// TIA Portal V17 export
// export: Created 2023-02-13T11:05:56.0459047Z, ExportSetting WithDefaults, DisplayName Totally Integrated Automation Portal, DisplayVersion V17, DisplayName TIA Portal Openness, DisplayVersion V17, DisplayName TIA Portal Teamcenter Gateway, DisplayVersion V17, DisplayName TIA Portal Version Control Interface, DisplayVersion V17, DisplayName SINAMICS Startdrive Advanced, DisplayVersion V17, DisplayName SINAMICS Startdrive G130, G150, S120, S150, SINAMICS MV, S210, DisplayVersion V17, DisplayName SINAMICS Startdrive G110M, G120, G120C, G120D, G120P, G115D, DisplayVersion V17, DisplayName STEP 7 Professional, DisplayVersion V17, DisplayName STEP 7 Safety, DisplayVersion V17, DisplayName WinCC Professional, DisplayVersion V17
VAR_GLOBAL   // PLC tag table "Tag table_1"
   "FT-02.01_Mass flow Value" AT %ID115 : Real;
   "FT-02.01_Mass flow Status" AT %IB119 : Byte;
   "FT-02.01_Volume flow Value" AT %ID120 : Real;
   "FT-02.01_Volume flow Status" AT %IB124 : Byte;
   "FT-02.01_Corrected volume flow Value" AT %ID125 : Real;
   "FT-02.01_Corrected volume flow Status" AT %IB129 : Byte;
   "FT-02.01_Density Value" AT %ID130 : Real;
   "FT-02.01_Density Status" AT %IB134 : Byte;
   "FT-02.01_Reference Density Value" AT %ID135 : Real;
   "FT-02.01_Reference Density Status" AT %IB139 : Byte;
   "FT-02.01_Temperature Value" AT %ID140 : Real;
   "FT-02.01_Temperature Status" AT %IB144 : Byte;
   "FT-02.01_Totalizer_1 Value" AT %ID145 : Real;
   "FT-02.01_Totalizer_1 Status" AT %IB149 : Byte;
   "FT-02.01_Totalizer_2 Value" AT %ID150 : Real;
   "FT-02.01_Totalizer_2 Status" AT %IB154 : Byte;
   "FT-02.01_Totalizer_3 Value" AT %ID155 : Real;
   "FT-02.01_Totalizer_3 Status" AT %IB159 : Byte;
   "FT-03.01_Mass flow Value" AT %ID160 : Real;
   "FT-03.01_Mass flow Status" AT %IB164 : Byte;
   "FT-03.01_Volume flow Value" AT %ID165 : Real;
   "FT-03.01_Volume flow Status" AT %IB169 : Byte;
   "FT-03.01_Corrected volume flow Value" AT %ID170 : Real;
   "FT-03.01_Corrected volume flow Status" AT %IB174 : Byte;
   "FT-03.01_Density Value" AT %ID175 : Real;
   "FT-03.01_Density Status" AT %IB179 : Byte;
   "FT-03.01_Reference Density Value" AT %ID180 : Real;
   "FT-03.01_Reference Density Status" AT %IB184 : Byte;
   "FT-03.01_Temperature Value" AT %ID185 : Real;
   "FT-03.01_Temperature Status" AT %IB189 : Byte;
   "FT-03.01_Totalizer_1 Value" AT %ID190 : Real;
   "FT-03.01_Totalizer_1 Status" AT %IB194 : Byte;
   "FT-03.01_Totalizer_2 Value" AT %ID195 : Real;
   "FT-03.01_Totalizer_2 Status" AT %IB199 : Byte;
   "FT-03.01_Totalizer_3 Value" AT %ID200 : Real;
   "FT-03.01_Totalizer_3 Status" AT %IB204 : Byte;
   "FT-04.01_Mass flow Value" AT %ID205 : Real;
   "FT-04.01_Mass flow Status" AT %IB209 : Byte;
   "FT-04.01_Volume flow Value" AT %ID210 : Real;
   "FT-04.01_Volume flow Status" AT %IB214 : Byte;
   "FT-04.01_Corrected volume flow Value" AT %ID215 : Real;
   "FT-04.01_Corrected volume flow Status" AT %IB219 : Byte;
   "FT-04.01_Density Value" AT %ID220 : Real;
   "FT-04.01_Density Status" AT %IB224 : Byte;
   "FT-04.01_Reference Density Value" AT %ID225 : Real;
   "FT-04.01_Reference Density Status" AT %IB229 : Byte;
   "FT-04.01_Temperature Value" AT %ID230 : Real;
   "FT-04.01_Temperature Status" AT %IB234 : Byte;
   "FT-04.01_Totalizer_1 Value" AT %ID235 : Real;
   "FT-04.01_Totalizer_1 Status" AT %IB239 : Byte;
   "FT-04.01_Totalizer_2 Value" AT %ID240 : Real;
   "FT-04.01_Totalizer_2 Status" AT %IB244 : Byte;
   "FT-04.01_Totalizer_3 Value" AT %ID245 : Real;
   "FT-04.01_Totalizer_3 Status" AT %IB249 : Byte;
   "FT-05.01_Mass flow Value" AT %ID250 : Real;
   "FT-05.01_Mass flow Status" AT %IB254 : Byte;
   "FT-05.01_Volume flow Value" AT %ID255 : Real;
   "FT-05.01_Volume flow Status" AT %IB259 : Byte;
   "FT-05.01_Corrected volume flow Value" AT %ID260 : Real;
   "FT-05.01_Corrected volume flow Status" AT %IB264 : Byte;
   "FT-05.01_Density Value" AT %ID265 : Real;
   "FT-05.01_Density Status" AT %IB269 : Byte;
   "FT-05.01_Reference Density Value" AT %ID270 : Real;
   "FT-05.01_Reference Density Status" AT %IB274 : Byte;
   "FT-05.01_Temperature Value" AT %ID275 : Real;
   "FT-05.01_Temperature Status" AT %IB279 : Byte;
   "FT-05.01_Totalizer_1 Value" AT %ID280 : Real;
   "FT-05.01_Totalizer_1 Status" AT %IB284 : Byte;
   "FT-05.01_Totalizer_2 Value" AT %ID285 : Real;
   "FT-05.01_Totalizer_2 Status" AT %IB289 : Byte;
   "FT-05.01_Totalizer_3 Value" AT %ID290 : Real;
   "FT-05.01_Totalizer_3 Status" AT %IB294 : Byte;
   "FT-06.01_Mass flow Value" AT %ID295 : Real;
   "FT-06.01_Mass flow Status" AT %IB299 : Byte;
   "FT-06.01_Volume flow Value" AT %ID300 : Real;
   "FT-06.01_Volume flow Status" AT %IB304 : Byte;
   "FT-06.01_Corrected volume flow Value" AT %ID305 : Real;
   "FT-06.01_Corrected volume flow Status" AT %IB309 : Byte;
   "FT-06.01_Density Value" AT %ID310 : Real;
   "FT-06.01_Density Status" AT %IB314 : Byte;
   "FT-06.01_Reference Density Value" AT %ID315 : Real;
   "FT-06.01_Reference Density Status" AT %IB319 : Byte;
   "FT-06.01_Temperature Value" AT %ID320 : Real;
   "FT-06.01_Temperature Status" AT %IB324 : Byte;
   "FT-06.01_Totalizer_1 Value" AT %ID325 : Real;
   "FT-06.01_Totalizer_1 Status" AT %IB329 : Byte;
   "FT-06.01_Totalizer_2 Value" AT %ID330 : Real;
   "FT-06.01_Totalizer_2 Status" AT %IB334 : Byte;
   "FT-06.01_Totalizer_3 Value" AT %ID335 : Real;
   "FT-06.01_Totalizer_3 Status" AT %IB339 : Byte;
   "FT-07.01_Mass flow Value" AT %ID340 : Real;
   "FT-07.01_Mass flow Status" AT %IB344 : Byte;
   "FT-07.01_Volume flow Value" AT %ID345 : Real;
   "FT-07.01_Volume flow Status" AT %IB349 : Byte;
   "FT-07.01_Corrected volume flow Value" AT %ID350 : Real;
   "FT-07.01_Corrected volume flow Status" AT %IB354 : Byte;
   "FT-07.01_Density Value" AT %ID355 : Real;
   "FT-07.01_Density Status" AT %IB359 : Byte;
   "FT-07.01_Reference Density Value" AT %ID360 : Real;
   "FT-07.01_Reference Density Status" AT %IB364 : Byte;
   "FT-07.01_Temperature Value" AT %ID365 : Real;
   "FT-07.01_Temperature Status" AT %IB369 : Byte;
   "FT-07.01_Totalizer_1 Value" AT %ID370 : Real;
   "FT-07.01_Totalizer_1 Status" AT %IB374 : Byte;
   "FT-07.01_Totalizer_2 Value" AT %ID375 : Real;
   "FT-07.01_Totalizer_2 Status" AT %IB379 : Byte;
   "FT-07.01_Totalizer_3 Value" AT %ID380 : Real;
   "FT-07.01_Totalizer_3 Status" AT %IB384 : Byte;
   "FT-08.01_Mass flow Value" AT %ID385 : Real;
   "FT-08.01_Mass flow Status" AT %IB389 : Byte;
   "FT-08.01_Volume flow Value" AT %ID390 : Real;
   "FT-08.01_Volume flow Status" AT %IB394 : Byte;
   "FT-08.01_Corrected volume flow Value" AT %ID395 : Real;
   "FT-08.01_Corrected volume flow Status" AT %IB399 : Byte;
   "FT-08.01_Density Value" AT %ID400 : Real;
   "FT-08.01_Density Status" AT %IB404 : Byte;
   "FT-08.01_Reference Density Value" AT %ID405 : Real;
   "FT-08.01_Reference Density Status" AT %IB409 : Byte;
   "FT-08.01_Temperature Value" AT %ID410 : Real;
   "FT-08.01_Temperature Status" AT %IB414 : Byte;
   "FT-08.01_Totalizer_1 Value" AT %ID415 : Real;
   "FT-08.01_Totalizer_1 Status" AT %IB419 : Byte;
   "FT-08.01_Totalizer_2 Value" AT %ID420 : Real;
   "FT-08.01_Totalizer_2 Status" AT %IB424 : Byte;
   "FT-08.01_Totalizer_3 Value" AT %ID425 : Real;
   "FT-08.01_Totalizer_3 Status" AT %IB429 : Byte;
   "FT-09.01_Mass flow Value" AT %ID430 : Real;
   "FT-09.01_Mass flow Status" AT %IB434 : Byte;
   "FT-09.01_Volume flow Value" AT %ID435 : Real;
   "FT-09.01_Volume flow Status" AT %IB439 : Byte;
   "FT-09.01_Corrected volume flow Value" AT %ID440 : Real;
   "FT-09.01_Corrected volume flow Status" AT %IB444 : Byte;
   "FT-09.01_Density Value" AT %ID445 : Real;
   "FT-09.01_Density Status" AT %IB449 : Byte;
   "FT-09.01_Reference Density Value" AT %ID450 : Real;
   "FT-09.01_Reference Density Status" AT %IB454 : Byte;
   "FT-09.01_Temperature Value" AT %ID455 : Real;
   "FT-09.01_Temperature Status" AT %IB459 : Byte;
   "FT-09.01_Totalizer_1 Value" AT %ID460 : Real;
   "FT-09.01_Totalizer_1 Status" AT %IB464 : Byte;
   "FT-09.01_Totalizer_2 Value" AT %ID465 : Real;
   "FT-09.01_Totalizer_2 Status" AT %IB469 : Byte;
   "FT-09.01_Totalizer_3 Value" AT %ID470 : Real;
   "FT-09.01_Totalizer_3 Status" AT %IB474 : Byte;
   "FT-10.01_Mass flow Value" AT %ID520 : Real;
   "FT-10.01_Mass flow Status" AT %IB524 : Byte;
   "FT-10.01_Volume flow Value" AT %ID525 : Real;
   "FT-10.01_Volume flow Status" AT %IB529 : Byte;
   "FT-10.01_Corrected volume flow Value" AT %ID530 : Real;
   "FT-10.01_Corrected volume flow Status" AT %IB534 : Byte;
   "FT-10.01_Density Value" AT %ID535 : Real;
   "FT-10.01_Density Status" AT %IB539 : Byte;
   "FT-10.01_Reference Density Value" AT %ID540 : Real;
   "FT-10.01_Reference Density Status" AT %IB544 : Byte;
   "FT-10.01_Temperature Value" AT %ID545 : Real;
   "FT-10.01_Temperature Status" AT %IB549 : Byte;
   "FT-10.01_Totalizer_1 Value" AT %ID550 : Real;
   "FT-10.01_Totalizer_1 Status" AT %IB554 : Byte;
   "FT-10.01_Totalizer_2 Value" AT %ID555 : Real;
   "FT-10.01_Totalizer_2 Status" AT %IB559 : Byte;
   "FT-10.01_Totalizer_3 Value" AT %ID560 : Real;
   "FT-10.01_Totalizer_3 Status" AT %IB564 : Byte;
   "FT-15.01_Mass flow Value" AT %ID475 : Real;
   "FT-15.01_Mass flow Status" AT %IB479 : Byte;
   "FT-15.01_Volume flow Value" AT %ID480 : Real;
   "FT-15.01_Volume flow Status" AT %IB484 : Byte;
   "FT-15.01_Corrected volume flow Value" AT %ID485 : Real;
   "FT-15.01_Corrected volume flow Status" AT %IB489 : Byte;
   "FT-15.01_Density Value" AT %ID490 : Real;
   "FT-15.01_Density Status" AT %IB494 : Byte;
   "FT-15.01_Reference Density Value" AT %ID495 : Real;
   "FT-15.01_Reference Density Status" AT %IB499 : Byte;
   "FT-15.01_Temperature Value" AT %ID500 : Real;
   "FT-15.01_Temperature Status" AT %IB504 : Byte;
   "FT-15.01_Totalizer_1 Value" AT %ID505 : Real;
   "FT-15.01_Totalizer_1 Status" AT %IB509 : Byte;
   "FT-15.01_Totalizer_2 Value" AT %ID510 : Real;
   "FT-15.01_Totalizer_2 Status" AT %IB514 : Byte;
   "FT-15.01_Totalizer_3 Value" AT %ID515 : Real;
   "FT-15.01_Totalizer_3 Status" AT %IB519 : Byte;
   "FT-22.01_Mass flow Value" AT %ID565 : Real;
   "FT-22.01_Mass flow Status" AT %IB569 : Byte;
   "FT-22.01_Volume flow Value" AT %ID570 : Real;
   "FT-22.01_Volume flow Status" AT %IB574 : Byte;
   "FT-22.01_Corrected volume flow Value" AT %ID575 : Real;
   "FT-22.01_Corrected volume flow Status" AT %IB579 : Byte;
   "FT-22.01_Density Value" AT %ID580 : Real;
   "FT-22.01_Density Status" AT %IB584 : Byte;
   "FT-22.01_Reference Density Value" AT %ID585 : Real;
   "FT-22.01_Reference Density Status" AT %IB589 : Byte;
   "FT-22.01_Temperature Value" AT %ID590 : Real;
   "FT-22.01_Temperature Status" AT %IB594 : Byte;
   "FT-22.01_Totalizer_1 Value" AT %ID595 : Real;
   "FT-22.01_Totalizer_1 Status" AT %IB599 : Byte;
   "FT-22.01_Totalizer_2 Value" AT %ID600 : Real;
   "FT-22.01_Totalizer_2 Status" AT %IB604 : Byte;
   "FT-22.01_Totalizer_3 Value" AT %ID605 : Real;
   "FT-22.01_Totalizer_3 Status" AT %IB609 : Byte;
   "FT-32.01_Mass flow Value" AT %ID610 : Real;
   "FT-32.01_Mass flow Status" AT %IB614 : Byte;
   "FT-32.01_Volume flow Value" AT %ID615 : Real;
   "FT-32.01_Volume flow Status" AT %IB619 : Byte;
   "FT-32.01_Corrected volume flow Value" AT %ID620 : Real;
   "FT-32.01_Corrected volume flow Status" AT %IB624 : Byte;
   "FT-32.01_Density Value" AT %ID625 : Real;
   "FT-32.01_Density Status" AT %IB629 : Byte;
   "FT-32.01_Reference Density Value" AT %ID630 : Real;
   "FT-32.01_Reference Density Status" AT %IB634 : Byte;
   "FT-32.01_Temperature Value" AT %ID635 : Real;
   "FT-32.01_Temperature Status" AT %IB639 : Byte;
   "FT-32.01_Totalizer_1 Value" AT %ID640 : Real;
   "FT-32.01_Totalizer_1 Status" AT %IB644 : Byte;
   "FT-32.01_Totalizer_2 Value" AT %ID645 : Real;
   "FT-32.01_Totalizer_2 Status" AT %IB649 : Byte;
   "FT-32.01_Totalizer_3 Value" AT %ID650 : Real;
   "FT-32.01_Totalizer_3 Status" AT %IB654 : Byte;
END_VAR
